# EPICS autosave request: GALIL/iocBoot/iocGALIL-IOC-01/GALIL_01_positions.req
file "GALIL_01_controller_positions.req" P=$(P),CCP=01
file "GALIL_01_controller_positions.req" P=$(P),CCP=02
file "GALIL_01_controller_positions.req" P=$(P),CCP=03
file "GALIL_01_controller_positions.req" P=$(P),CCP=04
file "GALIL_01_controller_positions.req" P=$(P),CCP=05
file "GALIL_01_controller_positions.req" P=$(P),CCP=06
file "GALIL_01_controller_positions.req" P=$(P),CCP=07
